Universal Robots PolyScope program: linear_push_on_taskboard.urp

Program linear_push_on_taskboard (installation=default directory=/programs createdIn=5.6.0.90886 lastSavedIn=5.6.0.90886 robotSerialNumber=20205500180)
Calibrated DH parameters: a=[0.000135, -0.030981, -0.334292, 0.000083, 0.000088, 0]; d=[0.162656, 258.79096, -331.603246, 72.945842, 0.099724, 0.099562]; alpha=[1.569535, 0.001639, 0.002824, 1.569633, -1.569323, 0]; deltaTheta=[0, 1.497881, -2.049261, 0.551379, 0, 0]
Robot Program (runOnlyOnce=true)
  MoveJ speed 60 deg/s, acceleration 80 deg/s^2 (useActiveTCP=false) tcp=gripper_140_tip; feature=Base
    Waypoint above_tb: TCP in base x=105.467 y=-471.694 z=337.495 mm, rx=2.2046 ry=-2.2187 rz=-0.0211 rad; joints [87.408, -92.681, 82.407, -79.697, -90.962, -92.28] deg; TCP offset x=0 y=0 z=220 mm, rx=0 ry=0 rz=0 rad
  URCap Gripper (Robotiq_Grippers, Robotiq Inc.) dataModel(position=100.0, force=100.0, speed=100.0, positionInDouble=100.0, forceInDouble=100.0, speedInDouble=100.0, slaveIds=[9], blocking=true)
  Force Frame feature=Base; selection=[0, 0, 1, 0, 0, 0]; wrench=[0, 0, -20, 0, 0, 0]; limitsForce=[0.15, 0.15, 0.01, 1.047198, 1.047198, 1.047198]; limitsMotion=[0.1, 0.1, 0.1, 0.349066, 0.349066, 0.349066]
    Wait Sleep waitTime=10
